FUNCTION_BLOCK CmdDAerationValvesBasic (* Basic Function Block Type *)
  (* Standard: 61499-2 *)
  (* Version 0.0, 8/9/2024, SESA713705, Schneider Electric, Template *)
  PACKAGE SE.Nereda;
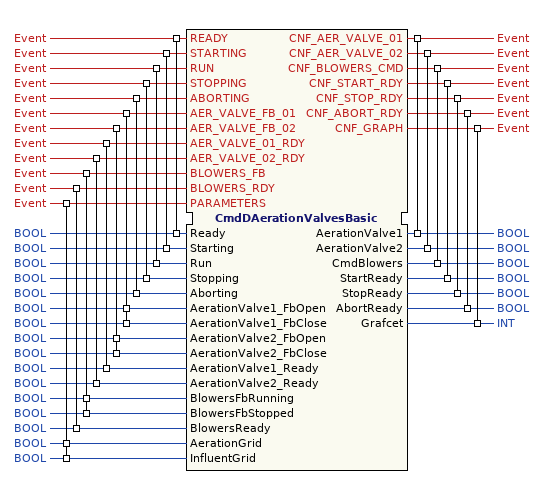
  EVENT_INPUT
    READY WITH Ready;
    STARTING WITH Starting;
    RUN WITH Run;
    STOPPING WITH Stopping;
    ABORTING WITH Aborting;
    AER_VALVE_FB_01 WITH AerationValve1_FbOpen, AerationValve1_FbClose;
    AER_VALVE_FB_02 WITH AerationValve2_FbOpen, AerationValve2_FbClose;
    AER_VALVE_01_RDY WITH AerationValve1_Ready;
    AER_VALVE_02_RDY WITH AerationValve2_Ready;
    BLOWERS_FB WITH BlowersFbRunning, BlowersFbStopped;
    BLOWERS_RDY WITH BlowersReady;
    PARAMETERS WITH AerationGrid, InfluentGrid;
  END_EVENT
  EVENT_OUTPUT
    CNF_AER_VALVE_01 WITH AerationValve1;
    CNF_AER_VALVE_02 WITH AerationValve2;
    CNF_BLOWERS_CMD WITH CmdBlowers;
    CNF_START_RDY WITH StartReady;
    CNF_STOP_RDY WITH StopReady;
    CNF_ABORT_RDY WITH AbortReady;
    CNF_GRAPH WITH Grafcet;
  END_EVENT
  VAR_INPUT
    Ready : BOOL;
    Starting : BOOL;
    Run : BOOL;
    Stopping : BOOL;
    Aborting : BOOL;
    AerationValve1_FbOpen : BOOL;
    AerationValve1_FbClose : BOOL;
    AerationValve2_FbOpen : BOOL;
    AerationValve2_FbClose : BOOL;
    AerationValve1_Ready : BOOL;
    AerationValve2_Ready : BOOL;
    BlowersFbRunning : BOOL;
    BlowersFbStopped : BOOL;
    BlowersReady : BOOL;
    AerationGrid : BOOL;
    InfluentGrid : BOOL;
  END_VAR
  VAR_OUTPUT
    AerationValve1 : BOOL; (* Aeration Grid Valve *)
    AerationValve2 : BOOL; (* Influent Grid Valve *)
    CmdBlowers : BOOL;
    StartReady : BOOL;
    StopReady : BOOL;
    AbortReady : BOOL;
    Grafcet : INT;
  END_VAR
  EC_STATES
    START; (* Initial State *)
    Ready : StopBlowers -> CNF_BLOWERS_CMD, -> CNF_START_RDY, -> CNF_ABORT_RDY, -> CNF_GRAPH;
    Starting : OpenValves -> CNF_AER_VALVE_01, -> CNF_AER_VALVE_02, -> CNF_STOP_RDY, -> CNF_ABORT_RDY, -> CNF_GRAPH;
    Run : RunBlowers -> CNF_BLOWERS_CMD, -> CNF_GRAPH;
    Stopping1 : StopBlowers -> CNF_BLOWERS_CMD, -> CNF_START_RDY, -> CNF_ABORT_RDY, -> CNF_GRAPH;
    Aborting1 : StopBlowers_WhenAborting -> CNF_BLOWERS_CMD, -> CNF_START_RDY, -> CNF_STOP_RDY, -> CNF_GRAPH;
    Abort;
    StopReady : StopReady -> CNF_STOP_RDY, -> CNF_GRAPH;
    Update : UpdateValvesState -> CNF_AER_VALVE_01, -> CNF_AER_VALVE_02, -> CNF_GRAPH;
    AbortReady : AbortReady -> CNF_ABORT_RDY, -> CNF_GRAPH;
    StartReday : StartReady -> CNF_START_RDY, -> CNF_GRAPH;
    Aborting2 : CloseAllValves -> CNF_AER_VALVE_01, -> CNF_AER_VALVE_02, -> CNF_GRAPH;
    Stopping2 : CloseAllValves -> CNF_AER_VALVE_01, -> CNF_AER_VALVE_02, -> CNF_GRAPH;
    CloseAll1 : CloseAllValves -> CNF_AER_VALVE_01, -> CNF_AER_VALVE_02, -> CNF_GRAPH;
    Open1stValve : Open1stValve -> CNF_AER_VALVE_01, -> CNF_AER_VALVE_02;
    Open2ndValve : UpdateValvesState -> CNF_AER_VALVE_01, -> CNF_AER_VALVE_02;
    NoParameter;
  END_STATES
  EC_TRANSITIONS
    START TO Ready := Ready AND (AerationValve1_FbOpen OR AerationValve2_FbOpen OR BlowersFbRunning);
    Ready TO CloseAll1 := BlowersFbStopped OR NOT BlowersReady;
    START TO Starting := STARTING AND Starting;
    Update TO Stopping1 := Stopping;
    START TO Aborting1 := ABORTING AND Aborting;
    Starting TO StartReday := (AerationValve1_FbOpen AND AerationGrid AND AerationValve2_FbClose AND NOT InfluentGrid) OR (AerationValve2_FbOpen AND InfluentGrid AND AerationValve1_FbClose AND NOT AerationGrid) OR (AerationValve1_FbOpen AND AerationGrid AND AerationValve2_FbOpen AND InfluentGrid);
    Abort TO Aborting1 := 1;
    Stopping1 TO Stopping2 := BlowersFbStopped;
    Run TO Update := BlowersFbRunning OR Stopping;
    Stopping1 TO Abort := ABORTING AND Aborting;
    Starting TO Abort := ABORTING AND Aborting;
    Run TO Abort := ABORTING AND Aborting;
    Update TO Abort := ABORTING AND Aborting;
    Aborting2 TO AbortReady := (AerationValve1_FbClose OR NOT AerationValve1_Ready) AND (AerationValve2_FbClose OR NOT AerationValve2_Ready);
    StopReady TO Abort := ABORTING AND Aborting;
    AbortReady TO START := 1;
    StopReady TO START := 1;
    StartReday TO Run := RUN AND Run = TRUE;
    Aborting1 TO Aborting2 := BlowersFbStopped OR NOT BlowersReady;
    Stopping2 TO StopReady := AerationValve1_FbClose AND AerationValve2_FbClose;
    CloseAll1 TO START := (AerationValve1_FbClose OR NOT AerationValve1_Ready) AND (AerationValve2_FbClose OR NOT AerationValve2_Ready);
    Starting TO Starting := PARAMETERS;
    Update TO NoParameter := PARAMETERS AND NOT AerationGrid AND NOT InfluentGrid;
    Open1stValve TO Open2ndValve := (AerationGrid AND AerationValve1_FbOpen) OR (InfluentGrid AND AerationValve2_FbOpen);
    Update TO Update := PARAMETERS AND (AerationGrid OR InfluentGrid);
    NoParameter TO Open1stValve := PARAMETERS AND (AerationGrid OR InfluentGrid);
    Open2ndValve TO Update := 1;
    Open1stValve TO Stopping1 := Stopping;
    NoParameter TO Stopping1 := Stopping;
    NoParameter TO Abort := ABORTING AND Aborting;
    Open1stValve TO Abort := ABORTING AND Aborting;
    StartReday TO Stopping1 := Stopping;
  END_TRANSITIONS
  ALGORITHM CloseAllValves IN ST:
;
IF Grafcet = 5 THEN
	Grafcet := 6;
ELSIF Grafcet = 8 THEN
	Grafcet := 9;
ELSIF Grafcet = 11 THEN
	Grafcet := 12;
END_IF;
AerationValve1 := FALSE;
AerationValve2 := FALSE;
  END_ALGORITHM
  ALGORITHM StartReady IN ST:
;
Grafcet := 2;
StartReady := TRUE;
  END_ALGORITHM
  ALGORITHM OpenValves IN ST:
;
Grafcet := 1;
StopReady := FALSE;
AbortReady := FALSE;

IF AerationGrid AND NOT InfluentGrid THEN
	AerationValve1 := TRUE;
	AerationValve2 := FALSE;

ELSIF NOT AerationGrid AND InfluentGrid THEN
	AerationValve1 := FALSE;
	AerationValve2 := TRUE;

ELSIF AerationGrid AND InfluentGrid THEN
	AerationValve1 := TRUE;
	AerationValve2 := TRUE;
END_IF;
  END_ALGORITHM
  ALGORITHM UpdateValvesState IN ST:
;
Grafcet := 4;
IF AerationGrid AND NOT InfluentGrid THEN
	AerationValve1 := TRUE;
	AerationValve2 := FALSE;

ELSIF NOT AerationGrid AND InfluentGrid THEN
	AerationValve1 := FALSE;
	AerationValve2 := TRUE;

ELSIF AerationGrid AND InfluentGrid THEN
	AerationValve1 := TRUE;
	AerationValve2 := TRUE;
END_IF;
  END_ALGORITHM
  ALGORITHM AbortReady IN ST:
;
Grafcet := 10;
AbortReady := TRUE;
  END_ALGORITHM
  ALGORITHM StopReady IN ST:
;
Grafcet := 7;
StopReady := TRUE;
  END_ALGORITHM
  ALGORITHM RunBlowers IN ST:
;
Grafcet := 3;
CmdBlowers := TRUE;
  END_ALGORITHM
  ALGORITHM StopBlowers IN ST:
;
IF Grafcet = 4 THEN
	Grafcet := 5;
ELSE
	Grafcet := 11;
END_IF;
CmdBlowers := FALSE;
StartReady := FALSE;
AbortReady := FALSE;
  END_ALGORITHM
  ALGORITHM StopBlowers_WhenAborting IN ST:
;
Grafcet := 8;
CmdBlowers := FALSE;
StartReady := FALSE;
StopReady := FALSE;
  END_ALGORITHM
  ALGORITHM Open1stValve IN ST:
;
IF AerationGrid AND NOT InfluentGrid THEN
	AerationValve1 := TRUE;

ELSIF NOT AerationGrid AND InfluentGrid THEN
	AerationValve2 := TRUE;

ELSIF AerationGrid AND InfluentGrid THEN
	AerationValve1 := TRUE;
	AerationValve2 := TRUE;
END_IF;
  END_ALGORITHM
END_FUNCTION_BLOCK
